DATA_BLOCK "DB_Wh_POL"
{ S7_Optimized_Access := 'FALSE' }
VERSION : 0.1
   STRUCT
      HMI_Word_spare : DWord;
      Tank : Array[1..10] of "UDT_Tank_Full";
   END_STRUCT;


BEGIN

END_DATA_BLOCK

